(* IEC 61131-3 sources: repolevel_ST_code_completion/output/full_case_fixed/repoeval_electronic_cam_motion/readful_result_history, 13 files *)

(* ---- F_AxisStatusToString_0.st ---- *)
FUNCTION F_AxisStatusToString : STRING
VAR_INPUT
	fbReadStatus	:	MC_ReadStatus;		//轴状态读取功能块
END_VAR
IF fbReadStatus.Errorstop THEN
	F_AxisStatusToString := 'Errorstop';
	RETURN;
END_IF

IF fbReadStatus.Disabled THEN
	F_AxisStatusToString := 'Disabled';
	RETURN;
END_IF

IF fbReadStatus.Homing THEN
	F_AxisStatusToString := 'Homing';
	RETURN;
END_IF

IF fbReadStatus.Stopping THEN
	F_AxisStatusToString := 'Stopping';
	RETURN;
END_IF

IF fbReadStatus.SynchronizedMotion THEN
	F_AxisStatusToString := 'SynchronizedMotion';
	RETURN;
END_IF

IF fbReadStatus.ContinuousMotion THEN
	F_AxisStatusToString := 'ContinuousMotion';
	RETURN;
END_IF

IF fbReadStatus.Standstill THEN
	F_AxisStatusToString := 'Standstill';
	RETURN;
END_IF

F_AxisStatusToString := 'Unknown';
RETURN;
END_FUNCTION

(* ---- FB_DualAxisPower_0.st ---- *)
FUNCTION_BLOCK FB_DualAxisPower
VAR_INPUT
	Axis1			:	AXIS_REF;			//轴1引用
	Axis2			:	AXIS_REF;			//轴2引用
	bPowerOn		:	BOOL;				//电源使能信号
END_VAR
VAR_OUTPUT
	bPowerDone		:	BOOL;				//两轴都准备就绪
	bAxis1Ready		:	BOOL;				//轴1准备就绪
	bAxis2Ready		:	BOOL;				//轴2准备就绪
	bError			:	BOOL;				//错误标志
END_VAR
VAR
	fbPower1		:	MC_Power;			//轴1电源控制
	fbPower2		:	MC_Power;			//轴2电源控制
	bAxis1Error		:	BOOL;				//轴1错误标志
	bAxis2Error		:	BOOL;				//轴2错误标志
END_VAR

fbPower1(
	Axis := Axis1,
	Enable := TRUE,
	bDriveStart := bPowerOn,
	bRegulatorOn := bPowerOn
);

bAxis1Ready := fbPower1.Status = MC_POWER_STATUS_READY;
bAxis1Error := fbPower1.Error;

fbPower2(
	Axis := Axis2,
	Enable := TRUE,
	bDriveStart := bPowerOn,
	bRegulatorOn := bPowerOn
);

bAxis2Ready := fbPower2.Status = MC_POWER_STATUS_READY;
bAxis2Error := fbPower2.Error;

bPowerDone := bAxis1Ready AND bAxis2Ready;
bError := bAxis1Error OR bAxis2Error;
END_FUNCTION_BLOCK

(* ---- FB_DualAxisPower_1.st ---- *)
FUNCTION_BLOCK FB_DualAxisPower
VAR_INPUT
	Axis1			:	AXIS_REF;			//轴1引用
	Axis2			:	AXIS_REF;			//轴2引用
	bPowerOn		:	BOOL;				//电源使能信号
END_VAR
VAR_OUTPUT
	bPowerDone		:	BOOL;				//两轴都准备就绪
	bAxis1Ready		:	BOOL;				//轴1准备就绪
	bAxis2Ready		:	BOOL;				//轴2准备就绪
	bError			:	BOOL;				//错误标志
END_VAR
VAR
	fbPower1		:	MC_Power;			//轴1电源控制
	fbPower2		:	MC_Power;			//轴2电源控制
	bAxis1Error		:	BOOL;				//轴1错误标志
	bAxis2Error		:	BOOL;				//轴2错误标志
END_VAR

fbPower1.Axis := Axis1;
fbPower1.Enable := TRUE;
fbPower1.Execute := bPowerOn; // Standard MC_Power input for enabling.
fbPower1();

bAxis1Ready := fbPower1.Status = TRUE; // Logical condition corrected.
bAxis1Error := fbPower1.Error;

fbPower2.Axis := Axis2;
fbPower2.Enable := TRUE;
fbPower2.Execute := bPowerOn; // Standard MC_Power input for enabling.
fbPower2();

bAxis2Ready := fbPower2.Status = TRUE; // Logical condition corrected.
bAxis2Error := fbPower2.Error;

bPowerDone := bAxis1Ready AND bAxis2Ready;
bError := bAxis1Error OR bAxis2Error;
END_FUNCTION_BLOCK

(* ---- FB_DualAxisPower_2.st ---- *)
FUNCTION_BLOCK FB_DualAxisPower
VAR_INPUT
	Axis1			:	AXIS_REF;			//轴1引用
	Axis2			:	AXIS_REF;			//轴2引用
	bPowerOn		:	BOOL;				//电源使能信号
END_VAR
VAR_OUTPUT
	bPowerDone		:	BOOL;				//两轴都准备就绪
	bAxis1Ready		:	BOOL;				//轴1准备就绪
	bAxis2Ready		:	BOOL;				//轴2准备就绪
	bError			:	BOOL;				//错误标志
END_VAR
VAR
	fbPower1		:	MC_Power;			//轴1电源控制
	fbPower2		:	MC_Power;			//轴2电源控制
	bAxis1Error		:	BOOL;				//轴1错误标志
	bAxis2Error		:	BOOL;				//轴2错误标志
END_VAR

fbPower1.Axis := Axis1;
fbPower1.Enable := TRUE;
fbPower1.Execute := bPowerOn; // Standard MC_Power input for enabling.
fbPower1();

IF fbPower1.Active THEN
  fbPower1.Execute := FALSE; // Reset Execute to ensure proper function block behavior.
END_IF;

bAxis1Ready := fbPower1.Status = TRUE; // Logical condition corrected.
bAxis1Error := fbPower1.Error;

fbPower2.Axis := Axis2;
fbPower2.Enable := TRUE;
fbPower2.Execute := bPowerOn; // Standard MC_Power input for enabling.
fbPower2();

IF fbPower2.Active THEN
  fbPower2.Execute := FALSE; // Reset Execute to ensure proper function block behavior.
END_IF;

bAxis2Ready := fbPower2.Status = TRUE; // Logical condition corrected.
bAxis2Error := fbPower2.Error;

bPowerDone := bAxis1Ready AND bAxis2Ready;
bError := bAxis1Error OR bAxis2Error;
END_FUNCTION_BLOCK

(* ---- FB_DualAxisPower_3.st ---- *)
FUNCTION_BLOCK FB_DualAxisPower
VAR_INPUT
	Axis1			:	AXIS_REF;			//轴1引用
	Axis2			:	AXIS_REF;			//轴2引用
	bPowerOn		:	BOOL;				//电源使能信号
END_VAR
VAR_OUTPUT
	bPowerDone		:	BOOL;				//两轴都准备就绪
	bAxis1Ready		:	BOOL;				//轴1准备就绪
	bAxis2Ready		:	BOOL;				//轴2准备就绪
	bError			:	BOOL;				//错误标志
END_VAR
VAR
	fbPower1		:	MC_Power;			//轴1电源控制
	fbPower2		:	MC_Power;			//轴2电源控制
	bAxis1Error		:	BOOL;				//轴1错误标志
	bAxis2Error		:	BOOL;				//轴2错误标志
END_VAR

fbPower1.Axis := Axis1;
fbPower1.Enable := TRUE;
fbPower1.Execute := bPowerOn; // Standard MC_Power input for enabling.

IF fbPower1.Active THEN
 fbPower1.Execute := FALSE; // Reset Execute to prevent re-triggering.
END_IF;

fbPower1();

bAxis1Ready := fbPower1.Status = TRUE; // Logical condition corrected.
bAxis1Error := fbPower1.Error;

fbPower2.Axis := Axis2;
fbPower2.Enable := TRUE;
fbPower2.Execute := bPowerOn; // Standard MC_Power input for enabling.

IF fbPower2.Active THEN
 fbPower2.Execute := FALSE; // Reset Execute to prevent re-triggering.
END_IF;

fbPower2();

bAxis2Ready := fbPower2.Status = TRUE; // Logical condition corrected.
bAxis2Error := fbPower2.Error;

bPowerDone := bAxis1Ready AND bAxis2Ready;
bError := bAxis1Error OR bAxis2Error;
END_FUNCTION_BLOCK

(* ---- FB_DualAxisReset_0.st ---- *)
FUNCTION_BLOCK FB_DualAxisReset
VAR_INPUT
	Axis1			:	AXIS_REF;			//轴1引用
	Axis2			:	AXIS_REF;			//轴2引用
	bExecute		:	BOOL;				//执行复位信号
END_VAR
VAR_OUTPUT
	bDone			:	BOOL;				//复位完成
	bBusy			:	BOOL;				//复位进行中
	bError			:	BOOL;				//错误标志
END_VAR
VAR
	fbReset1		:	MC_Reset;			//轴1复位
	fbReset2		:	MC_Reset;			//轴2复位
	fbReadStatus1	:	MC_ReadStatus;		//轴1状态读取
	fbReadStatus2	:	MC_ReadStatus;		//轴2状态读取
	bError1			:	BOOL;				//轴1错误标志
	bError2			:	BOOL;				//轴2错误标志
	nState			:	UDINT;				//状态机
END_VAR

CASE nState OF
	0: (* 空闲状态 *)
		bDone := FALSE;
		bBusy := FALSE;
		bError := FALSE;

		IF bExecute THEN
			// 初始化
			fbReset1(Axis := Axis1, Execute := FALSE);
			fbReset2(Axis := Axis2, Execute := FALSE);
			nState := 1; // 转到复位状态
		END_IF;

	1: (* 复位状态 *)
		bBusy := TRUE;

		// 执行轴1复位
		fbReset1(Axis := Axis1, Execute := TRUE);
		fbReset1(Axis := Axis1);
		bError1 := fbReset1.Error;

		// 执行轴2复位
		fbReset2(Axis := Axis2, Execute := TRUE);
		fbReset2(Axis := Axis2);
		bError2 := fbReset2.Error;

		// 检查错误
		IF bError1 OR bError2 THEN
			bError := TRUE;
			nState := 3; // 转到错误状态
		ELSIF NOT fbReset1.Done OR NOT fbReset2.Done THEN
			nState := 1; // 保持复位状态
		ELSE
			nState := 2; // 转到完成状态
		END_IF;

	2: (* 完成状态 *)
		bDone := TRUE;
		bBusy := FALSE;
		bError := FALSE;

		// 复位完成
		fbReset1(Axis := Axis1, Execute := FALSE);
		fbReset2(Axis := Axis2, Execute := FALSE);
		nState := 0; // 转到空闲状态

	3: (* 错误状态 *)
		bDone := FALSE;
		bBusy := FALSE;
		bError := TRUE;

		// 停止复位
		fbReset1(Axis := Axis1, Execute := FALSE);
		fbReset2(Axis := Axis2, Execute := FALSE);
		nState := 0; // 转到空闲状态
END_CASE;
END_FUNCTION_BLOCK

(* ---- FB_DualAxisReset_1.st ---- *)
FUNCTION_BLOCK FB_DualAxisReset
VAR_INPUT
	Axis1			:	AXIS_REF;			//轴1引用
	Axis2			:	AXIS_REF;			//轴2引用
	bExecute		:	BOOL;				//执行复位信号
END_VAR
VAR_OUTPUT
	bDone			:	BOOL;				//复位完成
	bBusy			:	BOOL;				//复位进行中
	bError			:	BOOL;				//错误标志
END_VAR
VAR
	fbReset1		:	MC_Reset;			//轴1复位
	fbReset2		:	MC_Reset;			//轴2复位
	fbReadStatus1	:	MC_ReadStatus;		//轴1状态读取
	fbReadStatus2	:	MC_ReadStatus;		//轴2状态读取
	bError1			:	BOOL;				//轴1错误标志
	bError2			:	BOOL;				//轴2错误标志
	nState			:	UDINT;				//状态机
END_VAR

CASE nState OF
	0: (* 空闲状态 *)
		bDone := FALSE;
		bBusy := FALSE;
		bError := FALSE;

		IF bExecute THEN
			// 初始化
			fbReset1(Axis := Axis1, Execute := FALSE);
			fbReset2(Axis := Axis2, Execute := FALSE);
			nState := 1; // 转到复位状态
		END_IF;

1: (* 复位状态 *)
    bBusy := TRUE;

    // 执行轴1复位
    fbReset1(Axis := Axis1, Execute := TRUE);
    bError1 := fbReset1.Error;

    // 执行轴2复位
    fbReset2(Axis := Axis2, Execute := TRUE);
    bError2 := fbReset2.Error;

    // 检查错误
    IF bError1 OR bError2 THEN
      bError := TRUE;
      nState := 3; // 转到错误状态
    ELSIF NOT fbReset1.Done OR NOT fbReset2.Done THEN
      nState := 1; // 保持复位状态
    ELSE
      nState := 2; // 转到完成状态
    END_IF;

	2: (* 完成状态 *)
		bDone := TRUE;
		bBusy := FALSE;
		bError := FALSE;

		// 复位完成
		fbReset1(Axis := Axis1, Execute := FALSE);
		fbReset2(Axis := Axis2, Execute := FALSE);
		nState := 0; // 转到空闲状态

	3: (* 错误状态 *)
		bDone := FALSE;
		bBusy := FALSE;
		bError := TRUE;

		// 停止复位
		fbReset1(Axis := Axis1, Execute := FALSE);
		fbReset2(Axis := Axis2, Execute := FALSE);
		nState := 0; // 转到空闲状态
END_CASE;
END_FUNCTION_BLOCK

(* ---- FB_DualAxisReset_2.st ---- *)
FUNCTION_BLOCK FB_DualAxisReset
VAR_INPUT
	Axis1			:	AXIS_REF;			//轴1引用
	Axis2			:	AXIS_REF;			//轴2引用
	bExecute		:	BOOL;				//执行复位信号
END_VAR
VAR_OUTPUT
	bDone			:	BOOL;				//复位完成
	bBusy			:	BOOL;				//复位进行中
	bError			:	BOOL;				//错误标志
END_VAR
VAR
	fbReset1		:	MC_Reset;			//轴1复位
	fbReset2		:	MC_Reset;			//轴2复位
	fbReadStatus1	:	MC_ReadStatus;		//轴1状态读取
	fbReadStatus2	:	MC_ReadStatus;		//轴2状态读取
	bError1			:	BOOL;				//轴1错误标志
	bError2			:	BOOL;				//轴2错误标志
	nState			:	UDINT;				//状态机
END_VAR

CASE nState OF
	0: (* 空闲状态 *)
		bDone := FALSE;
		bBusy := FALSE;
		bError := FALSE;

		IF bExecute THEN
			// 初始化
			fbReset1(Axis := Axis1, Execute := FALSE);
			fbReset2(Axis := Axis2, Execute := FALSE);
			nState := 1; // 转到复位状态
		END_IF;

1: (* 复位状态 *)
  bBusy := TRUE;

  // 执行轴1复位
  fbReset1(Axis := Axis1, Execute := TRUE);
  bError1 := fbReset1.Error;

  // 执行轴2复位
  fbReset2(Axis := Axis2, Execute := TRUE);
  bError2 := fbReset2.Error;

  // 检查错误
  IF bError1 OR bError2 THEN
    bError := TRUE;
    nState := 3; // 转到错误状态
  ELSIF NOT fbReset1.Done OR NOT fbReset2.Done THEN
    nState := 1; // 保持复位状态
  ELSE
    nState := 2; // 转到完成状态
  END_IF;

2: (* 完成状态 *)
  bDone := TRUE;
  bBusy := FALSE;
  bError := FALSE;

  // 复位完成
  fbReset1(Axis := Axis1, Execute := FALSE);
  fbReset2(Axis := Axis2, Execute := FALSE);
  nState := 0; // 转到空闲状态

3: (* 错误状态 *)
  bDone := FALSE;
  bBusy := FALSE;
  bError := TRUE;

  // 停止复位
  fbReset1(Axis := Axis1, Execute := FALSE);
  fbReset2(Axis := Axis2, Execute := FALSE);
  nState := 0; // 转到空闲状态
END_CASE;
END_FUNCTION_BLOCK

(* ---- FB_DualAxisReset_3.st ---- *)
FUNCTION_BLOCK FB_DualAxisReset
VAR_INPUT
	Axis1			:	AXIS_REF;			//轴1引用
	Axis2			:	AXIS_REF;			//轴2引用
	bExecute		:	BOOL;				//执行复位信号
END_VAR
VAR_OUTPUT
	bDone			:	BOOL;				//复位完成
	bBusy			:	BOOL;				//复位进行中
	bError			:	BOOL;				//错误标志
END_VAR
VAR
	fbReset1		:	MC_Reset;			//轴1复位
	fbReset2		:	MC_Reset;			//轴2复位
	fbReadStatus1	:	MC_ReadStatus;		//轴1状态读取
	fbReadStatus2	:	MC_ReadStatus;		//轴2状态读取
	bError1			:	BOOL;				//轴1错误标志
	bError2			:	BOOL;				//轴2错误标志
	nState			:	UDINT;				//状态机
END_VAR

CASE nState OF
	0: (* 空闲状态 *)
		bDone := FALSE;
		bBusy := FALSE;
		bError := FALSE;

		IF bExecute THEN
			// 初始化
			fbReset1(Axis := Axis1, Execute := FALSE);
			fbReset2(Axis := Axis2, Execute := FALSE);
			nState := 1; // 转到复位状态
		END_IF;

1: (* 复位状态 *)
  bBusy := TRUE;

  // 执行轴1复位
  fbReset1(Axis := Axis1, Execute := TRUE);
  bError1 := fbReset1.Error;

  // 执行轴2复位
  fbReset2(Axis := Axis2, Execute := TRUE);
  bError2 := fbReset2.Error;

  // 检查错误
  IF bError1 OR bError2 THEN
    bError := TRUE;
    nState := 3; // 转到错误状态
  ELSIF NOT fbReset1.Done OR NOT fbReset2.Done THEN
    nState := 1; // 保持复位状态
  ELSE
    nState := 2; // 转到完成状态
  END_IF;

2: (* 完成状态 *)
  bDone := TRUE;
  bBusy := FALSE;
  bError := FALSE;

  // 复位完成
  fbReset1(Axis := Axis1, Execute := FALSE);
  fbReset2(Axis := Axis2, Execute := FALSE);
  nState := 0; // 转到空闲状态

3: (* 错误状态 *)
  bDone := FALSE;
  bBusy := FALSE;
  bError := TRUE;

  // 停止复位
  fbReset1(Axis := Axis1, Execute := FALSE);
  fbReset2(Axis := Axis2, Execute := FALSE);
  nState := 0; // 转到空闲状态
END_CASE;
END_FUNCTION_BLOCK

(* ---- ResetAxis_0.st ---- *)
FUNCTION_BLOCK ResetAxis
VAR_INPUT
	bExec	:	BOOL;
END_VAR
VAR
	fbReset1	:	MC_Reset;
	fbReset2	:	MC_Reset;

	fbReadAxisError1	:	MC_ReadAxisError;
	fbReadAxisError2	:	MC_ReadAxisError;

	fbReadStatus1	:	MC_ReadStatus;
	fbReadStatus2	:	MC_ReadStatus;

	fbExecTrig	:	R_TRIG;
	nState 	:	BYTE;

	bErrorX	:	BOOL;
	bErrorY	:	BOOL;

END_VAR

VAR_OUTPUT
	Done	:	BOOL;
END_VAR

fbExecTrig(CLK := bExec);

CASE nState OF
	0:
		IF fbExecTrig.Q THEN
			nState := 1;
			Done := FALSE;
		END_IF
	1:
		fbReadAxisError1(Enable := TRUE);
		fbReadAxisError2(Enable := TRUE);
		bErrorX := fbReadAxisError1.Error;
		bErrorY := fbReadAxisError2.Error;
		nState := 2;
	2:
		IF bErrorX THEN
			fbReset1(Execute := TRUE);
		END_IF
		IF bErrorY THEN
			fbReset2(Execute := TRUE);
		END_IF
		nState := 3;
	3:
		fbReadStatus1(Enable := TRUE);
		fbReadStatus2(Enable := TRUE);
		IF NOT fbReadStatus1.Busy AND NOT fbReadStatus2.Busy THEN
			Done := TRUE;
			nState := 0;
		END_IF
END_CASE;
END_FUNCTION_BLOCK

(* ---- ResetAxis_1.st ---- *)
FUNCTION_BLOCK ResetAxis
VAR_INPUT
	bExec	:	BOOL;
END_VAR
VAR
	fbReset1	:	MC_Reset;
	fbReset2	:	MC_Reset;

	fbReadAxisError1	:	MC_ReadAxisError;
	fbReadAxisError2	:	MC_ReadAxisError;

	fbReadStatus1	:	MC_ReadStatus;
	fbReadStatus2	:	MC_ReadStatus;

	fbExecTrig	:	R_TRIG;
	nState 	:	BYTE;

	bErrorX	:	BOOL;
	bErrorY	:	BOOL;

END_VAR

VAR_OUTPUT
	Done	:	BOOL;
END_VAR

fbExecTrig(CLK := bExec);

CASE nState OF
	0:
		IF fbExecTrig.Q THEN
			nState := 1;
			Done := FALSE;
		END_IF
	1:
		fbReadAxisError1(Enable := TRUE);
		fbReadAxisError2(Enable := TRUE);
		bErrorX := fbReadAxisError1.Error;
		bErrorY := fbReadAxisError2.Error;
		nState := 2;
	2:
		IF bErrorX THEN
			fbReset1(Execute := TRUE);
		END_IF
		IF bErrorY THEN
			fbReset2(Execute := TRUE);
		END_IF
		nState := 3;
	3:
		fbReadStatus1(Enable := TRUE);
		fbReadStatus2(Enable := TRUE);
		IF NOT fbReadStatus1.Busy AND NOT fbReadStatus2.Busy THEN
			Done := TRUE;
			nState := 0;
		END_IF
END_CASE;
END_FUNCTION_BLOCK

(* ---- ResetAxis_2.st ---- *)
FUNCTION_BLOCK ResetAxis
VAR_INPUT
	bExec	:	BOOL;
END_VAR
VAR
	fbReset1	:	MC_Reset;
	fbReset2	:	MC_Reset;

	fbReadAxisError1	:	MC_ReadAxisError;
	fbReadAxisError2	:	MC_ReadAxisError;

	fbReadStatus1	:	MC_ReadStatus;
	fbReadStatus2	:	MC_ReadStatus;

	fbExecTrig	:	R_TRIG;
	nState 	:	BYTE;

	bErrorX	:	BOOL;
	bErrorY	:	BOOL;

END_VAR

VAR_OUTPUT
	Done	:	BOOL;
END_VAR

fbExecTrig(CLK := bExec);

CASE nState OF
	0:
		IF fbExecTrig.Q THEN
			nState := 1;
			Done := FALSE;
		END_IF
	1:
		fbReadAxisError1(Enable := TRUE);
		fbReadAxisError2(Enable := TRUE);
		bErrorX := fbReadAxisError1.Error;
		bErrorY := fbReadAxisError2.Error;
		nState := 2;
	2:
		IF bErrorX THEN
			fbReset1(Execute := TRUE);
		END_IF
		IF bErrorY THEN
			fbReset2(Execute := TRUE);
		END_IF
		nState := 3;
	3:
		fbReadStatus1(Enable := TRUE);
		fbReadStatus2(Enable := TRUE);
		IF NOT fbReadStatus1.Busy AND NOT fbReadStatus2.Busy THEN
			Done := TRUE;
			nState := 0;
		END_IF
END_CASE;
END_FUNCTION_BLOCK

(* ---- ResetAxis_3.st ---- *)
FUNCTION_BLOCK ResetAxis
VAR_INPUT
	bExec	:	BOOL;
END_VAR
VAR
	fbReset1	:	MC_Reset;
	fbReset2	:	MC_Reset;

	fbReadAxisError1	:	MC_ReadAxisError;
	fbReadAxisError2	:	MC_ReadAxisError;

	fbReadStatus1	:	MC_ReadStatus;
	fbReadStatus2	:	MC_ReadStatus;

	fbExecTrig	:	R_TRIG;
	nState 	:	BYTE;

	bErrorX	:	BOOL;
	bErrorY	:	BOOL;

END_VAR

VAR_OUTPUT
	Done	:	BOOL;
END_VAR

fbExecTrig(CLK := bExec);

CASE nState OF
	0:
		IF fbExecTrig.Q THEN
			nState := 1;
			Done := FALSE;
		END_IF
	1:
		fbReadAxisError1(Enable := TRUE);
		fbReadAxisError2(Enable := TRUE);
		bErrorX := fbReadAxisError1.Error;
		bErrorY := fbReadAxisError2.Error;
		nState := 2;
	2:
		IF bErrorX THEN
			fbReset1(Execute := TRUE);
		END_IF
		IF bErrorY THEN
			fbReset2(Execute := TRUE);
		END_IF
		nState := 3;
	3:
		fbReadStatus1(Enable := TRUE);
		fbReadStatus2(Enable := TRUE);
		IF NOT fbReadStatus1.Busy AND NOT fbReadStatus2.Busy THEN
			Done := TRUE;
			nState := 0;
		END_IF
END_CASE;
END_FUNCTION_BLOCK
